{attribute 'qualified_only'}
VAR_GLOBAL
	bSimRunning : BOOL;
	fSimulationTime : LREAL;
	fCylinderVelocity : LREAL;
	fCylinderPosition : LREAL;
END_VAR

(* stored: Version 1.1.0.1, ProductVersion 3.1.4024.10
   GVL Outputs: Id {ef6fc48f-0dd8-459d-85d3-31e8a9c5d05f} *)
